RoboDK station: workstation_tire_stack_unstack.rdk

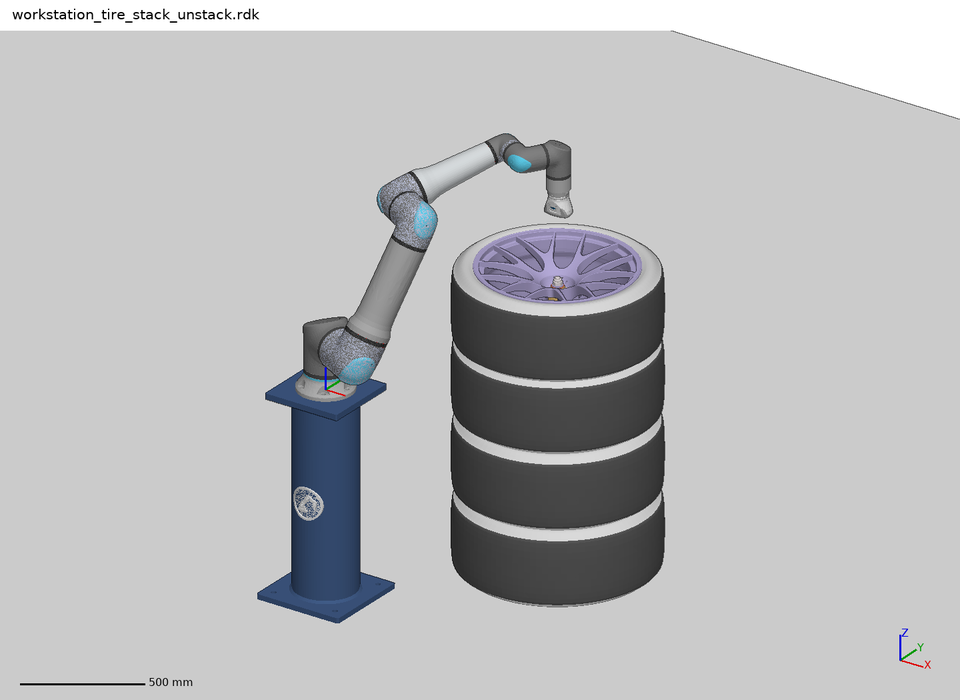
[picture v0: the station drawn from its stored meshes, robots at their saved joint values, targets as dots, program paths as lines]
Station New Station (15555555) (saved by RoboDK 5.2.4). Poses are relative to the parent item; angles as X-Y-Z fixed-axis rotations.
  - frame UR30 Base at (0, 0, 910) mm
    - robot UR30 (model UR20): 6 axes
        modified DH rows (alpha deg, a mm, theta deg, d mm): 0, 0, 0, 236.2; 90, 0, -180, 0; 0, 636.8, 0, 0; 0, 505.7, 0, 201.9; -90, 0, 0, 159.4; 90, 0, 0, 154.8
        joint limits [-360, -360, -360, -360, -360, -360] to [360, 360, 360, 360, 360, 360]; home [0, -90, -90, 0, 90, 0]; saved at [60.449, -116.881, -47.119, 254.08, -269.955, 330.449]
      - robot SCHUNK Co-act Gripper: 1 axes
          joint limits [0] to [40]; home [0]; saved at [0]
      - tool Tool, TCP at (0, 0, 200) mm
  - object Pedestal H36in (Type 1) at (0, 0, 0) mm, size 400 x 400 x 914.4 mm, geometry from Pedestal-H36in-Type-1.sld
  - object plane at (0, 0, 0) mm, size 10000 x 10000 x 0 mm, geometry from plane.obj
  - object T3 at (520, 290, 2070) mm, size 338.9 x 855.2 x 855.2 mm, geometry from Wheel BBS Michelin N260121.obj
  - object T2 at (520, 290, 1730) mm, size 338.9 x 855.2 x 855.2 mm, geometry from Wheel BBS Michelin N260121.obj
  - program Prog1 (4 instructions, listed below)
  - object T1 at (520, 290, 1390) mm, size 338.9 x 855.2 x 855.2 mm, geometry from Wheel BBS Michelin N260121.obj
  - object T4 at (520, 290, 2390) mm, size 338.9 x 855.2 x 855.2 mm, geometry from Wheel BBS Michelin N260121.obj

--- program Prog1 (robot UR30) ---
  Replace T1
  Replace T2
  Replace T3
  Replace T4
